TYPE TFRullieraManCmd :
STRUCT
	Ax 					: TFAxManCmd;
	ResetModulo 		: BOOL;
	Ax2 				: TFAxManCmd;
	AbilitaCmdTandemRulliere	: BOOL;
END_STRUCT
END_TYPE

(* stored: Version 1.1.0.1, ProductVersion 3.1.4024.11
   DUT TFRullieraManCmd: Id {9b154f33-7bce-4bb7-b7a6-c2ab5ae0b711} *)
